(* CODESYS project ManualControl.xml

Project tree, tasks and I/O mapping:
  function block ManualControl [LD]
*)

// ManualControl
FUNCTION_BLOCK ManualControl
VAR_OUTPUT
	TriggerAgitate: BOOL;
	DoorLock: BOOL;
	MakeIce: BOOL;
	OpenHeatSeal: BOOL;
	CloseHeatSeal: BOOL;
END_VAR

// NETWORK 1

END_FUNCTION_BLOCK
